(* CODESYS project ai_oven_00_90.project
   Description: Receives some incoming messages and echoes them with CAN-ID +1
   Author: 3S - Smart Software Solutions GmbH
   Version: 1.0.0.0
   Title: CAN Bus API Example
   Company: 3S - Smart Software Solutions GmbH

Project tree, tasks and I/O mapping:
  xLH : CODESYS Control for Raspberry Pi 64 SL, CODESYS, order no. 2302000009, version 4.18.0.0
    application app
      libraries: Standard, 3.5.18.0 (System); Memory, * (3S - Smart Software Solutions GmbH); Util, 3.5.21.0 (System); VisuDialogs, * (System); CAA Tick Extern, 3.5.17.0 (CAA Technical Workgroup); SysTime, 3.5.17.0 (System); CmpIecTask, * (System); StringUtils, 3.5.20.0 (System); MQTT Client SL, 1.12.0.0 (CODESYS)
      task MAIN_TASK (cyclic, interval 20 ms, priority 0) calls MAIN
      task VISU_TASK (cyclic, interval 100 ms, priority 31) calls VisuElems.Visu_Prg
      visualisation Visualization
      program MAIN [ST]
      Symbols
    SoftMotion General Axis Pool
    GPIOs_A_B : GPIOs B+/Pi2, CODESYS, version 4.18.0.0
        unmapped channels: digital inputs (GPIO0..GPIO31), digital outputs (GPIO0..GPIO31)
    Onewire
    Camera device
      <Leer>
    SPI
    I²C
  libraries: VisuSymbols, 4.5.0.0 (System); DepictorBase, 1.2.0.0 (CODESYS)
  text list GlobalTextList
*)

// xLH/app/MAIN
PROGRAM MAIN
VAR
	rOvenTemperatureSetpoint: REAL;
	rDummy: REAL;
END_VAR

rDummy := rOvenTemperatureSetpoint;

END_PROGRAM

// xLH/app/Visualization
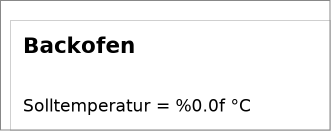
VISUALIZATION Visualization  // 331x131
    Rectangle (10,20 321x111)
    Rectangle (20,20 301x51), "Backofen"
    Rectangle (20,80 300x51), "Solltemperatur = %0.0f °C", text variable: MAIN.rOvenTemperatureSetpoint
END_VISUALIZATION
